Staubli VAL3: tableSpeed.pgx

public program tableSpeed(num x_nSpeedCase (dimensions=1))
  local num l_nNum
  local num l_nNum2
begin
  l_nNum=roundDown(x_nSpeedCase/16)
  l_nNum2=x_nSpeedCase%16
  switch l_nNum
    //0-15
    case 0
      call speedCase0_15(l_nNum2)
    break
    //16-31
    case 1
      call speedCase0_15(l_nNum2)

      dioSet(doB_4_speed,1)
    break
    //32-63
    //32-47
    case 2
      call speedCase0_15(l_nNum2)
      dioSet(doB_5_speed,1)
    break
    //48-63
    case 3
      call speedCase0_15(l_nNum2)

      dioSet(doB_4_speed,1)
      dioSet(doB_5_speed,1)
    break
    //    //64-127
    //    //64-79
    //    case 4
    //      call speedCase0_15(l_nNum2)
    //      dioSet(doB_6_speed,1)
    //    break
    //    case 5
    //      call speedCase0_15(l_nNum2)
    //      dioSet(doB_4_speed,1)
    //      dioSet(doB_6_speed,1)
    //    break
    //    //80-95
    //    case 6
    //      call speedCase0_15(l_nNum2)
    //      dioSet(doB_5_speed,1)
    //      dioSet(doB_6_speed,1)
    //    break
    //    //96-127
    //    case 7
    //      call speedCase0_15(l_nNum2)
    //      dioSet(doB_4_speed,1)
    //      dioSet(doB_5_speed,1)
    ////      dioSet(doB_6_speed,1)
    //    break
    //    //128-255
    //    //128-143
    //    case 8
    //      call speedCase0_15(l_nNum2)
    ////      dioSet(doB_7_speed,1)
    //    break
    //      //144-159
    //    case 9
    //      call speedCase0_15(l_nNum2)
    //      dioSet(doB_4_speed,1)
    ////      dioSet(doB_7_speed,1)
    //    break
    //      //160-175
    //    case 10
    //      call speedCase0_15(l_nNum2)
    //      dioSet(doB_5_speed,1)
    ////      dioSet(doB_7_speed,1)
    //    break
    //      //176-191
    //    case 11
    //      call speedCase0_15(l_nNum2)
    //      dioSet(doB_4_speed,1)
    //      dioSet(doB_5_speed,1)
    ////      dioSet(doB_7_speed,1)
    //    break
    //      //192-207
    //    case 12
    //      call speedCase0_15(l_nNum2)
    ////      dioSet(doB_6_speed,1)
    ////      dioSet(doB_7_speed,1)
    //    break
    //    //208-223
    //    case 13
    //      call speedCase0_15(l_nNum2)
    //      dioSet(doB_4_speed,1)
    ////      dioSet(doB_6_speed,1)
    ////      dioSet(doB_7_speed,1)
    //    break
    //      //224-239
    //    case 14
    //      call speedCase0_15(l_nNum2)
    //      dioSet(doB_5_speed,1)
    ////      dioSet(doB_6_speed,1)
    ////      dioSet(doB_7_speed,1)
    //    break
    //      //240-255
    //    case 15
    //      call speedCase0_15(l_nNum2)
    //      dioSet(doB_4_speed,1)
    //      dioSet(doB_5_speed,1)
    ////      dioSet(doB_6_speed,1)
    ////      dioSet(doB_7_speed,1)
    //    break
  endSwitch











end
